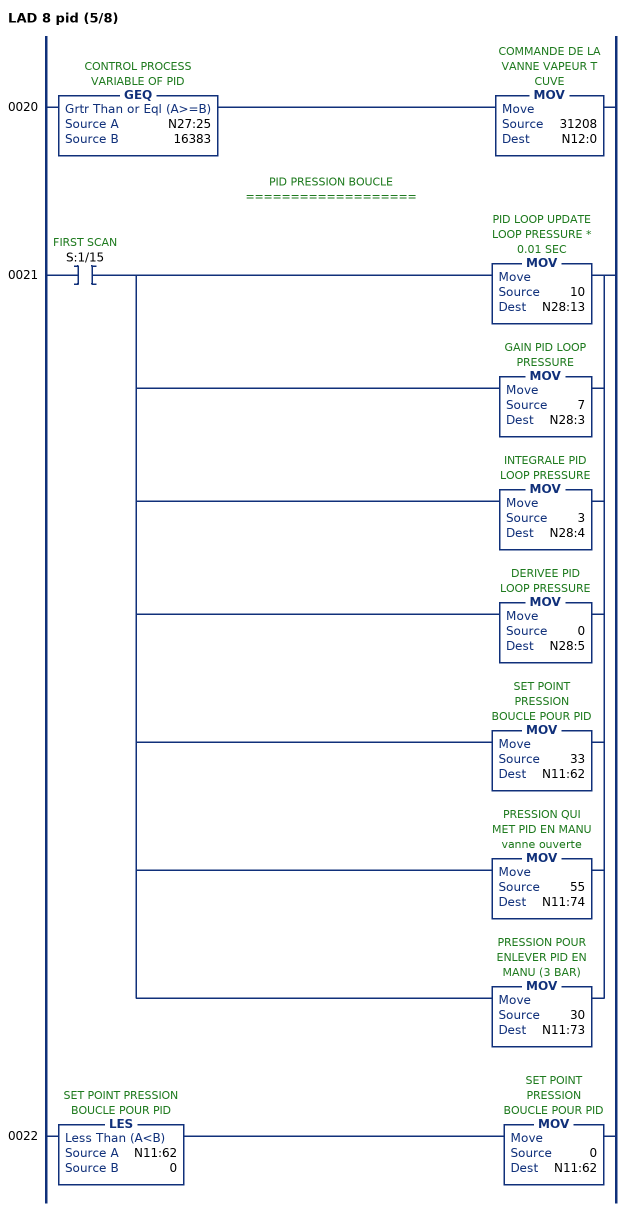
% Rung: 20 %
SOR GEQ N27:25 16383 MOV 31208 N12:0 EOR
%   N27:25  "CONTROL PROCESS VARIABLE OF PID" %
%   N12:0  "COMMANDE DE LA VANNE VAPEUR T CUVE" %
% Rung: 21 %
% PID PRESSION BOUCLE
% =================== %
SOR XIC S:1/15 BST MOV 10 N28:13 NXB MOV 7 N28:3 NXB MOV 3 N28:4 NXB MOV 0 N28:5 NXB MOV 33 N11:62 NXB MOV 55 N11:74 NXB MOV 30 N11:73 BND EOR
%   S:1/15  "FIRST SCAN" %
%   N28:13  "PID LOOP UPDATE LOOP PRESSURE * 0.01 SEC" %
%   N28:3  "GAIN PID LOOP PRESSURE" %
%   N28:4  "INTEGRALE PID LOOP PRESSURE" %
%   N28:5  "DERIVEE PID LOOP PRESSURE" %
%   N11:62  "SET POINT PRESSION BOUCLE POUR PID" %
%   N11:74  "PRESSION QUI MET PID EN MANU vanne ouverte" %
%   N11:73  "PRESSION POUR ENLEVER PID EN MANU (3 BAR)" %
% Rung: 22 %
SOR LES N11:62 0 MOV 0 N11:62 EOR
%   N11:62  "SET POINT PRESSION BOUCLE POUR PID" %

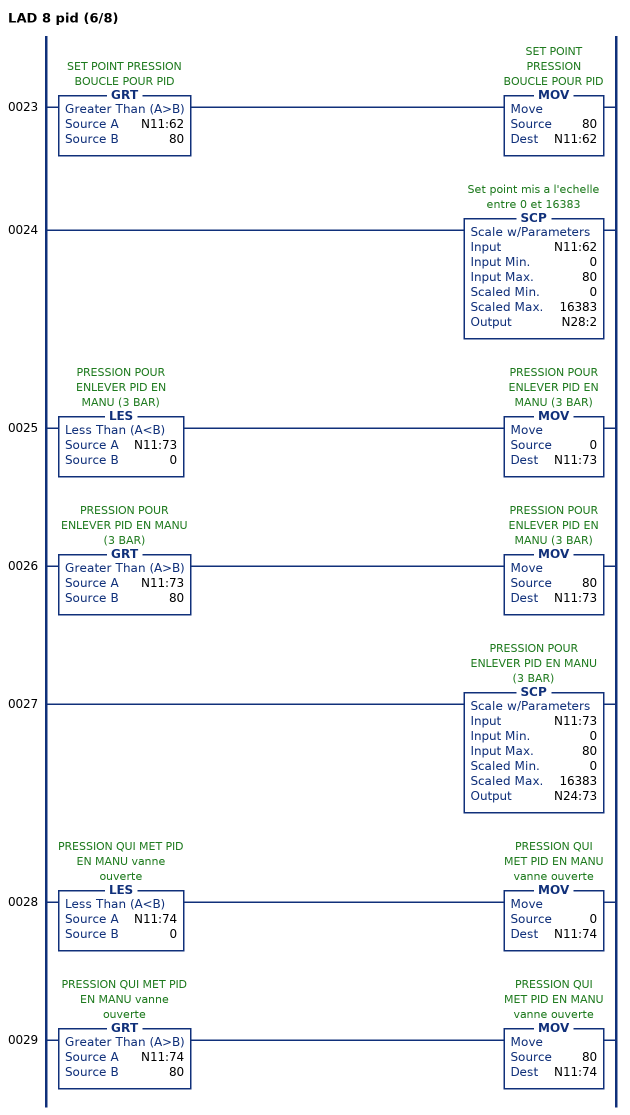
% Rung: 23 %
SOR GRT N11:62 80 MOV 80 N11:62 EOR
%   N11:62  "SET POINT PRESSION BOUCLE POUR PID" %
% Rung: 24 %
SOR SCP N11:62 0 80 0 16383 N28:2 EOR
%   N11:62  "SET POINT PRESSION BOUCLE POUR PID" %
%   N28:2  "Set point mis a l'echelle entre 0 et 16383" %
% Rung: 25 %
SOR LES N11:73 0 MOV 0 N11:73 EOR
%   N11:73  "PRESSION POUR ENLEVER PID EN MANU (3 BAR)" %
% Rung: 26 %
SOR GRT N11:73 80 MOV 80 N11:73 EOR
%   N11:73  "PRESSION POUR ENLEVER PID EN MANU (3 BAR)" %
% Rung: 27 %
SOR SCP N11:73 0 80 0 16383 N24:73 EOR
%   N11:73  "PRESSION POUR ENLEVER PID EN MANU (3 BAR)" %
%   N24:73  "PRESSION POUR ENLEVER PID EN MANU (3 BAR)" %
% Rung: 28 %
SOR LES N11:74 0 MOV 0 N11:74 EOR
%   N11:74  "PRESSION QUI MET PID EN MANU vanne ouverte" %
% Rung: 29 %
SOR GRT N11:74 80 MOV 80 N11:74 EOR
%   N11:74  "PRESSION QUI MET PID EN MANU vanne ouverte" %

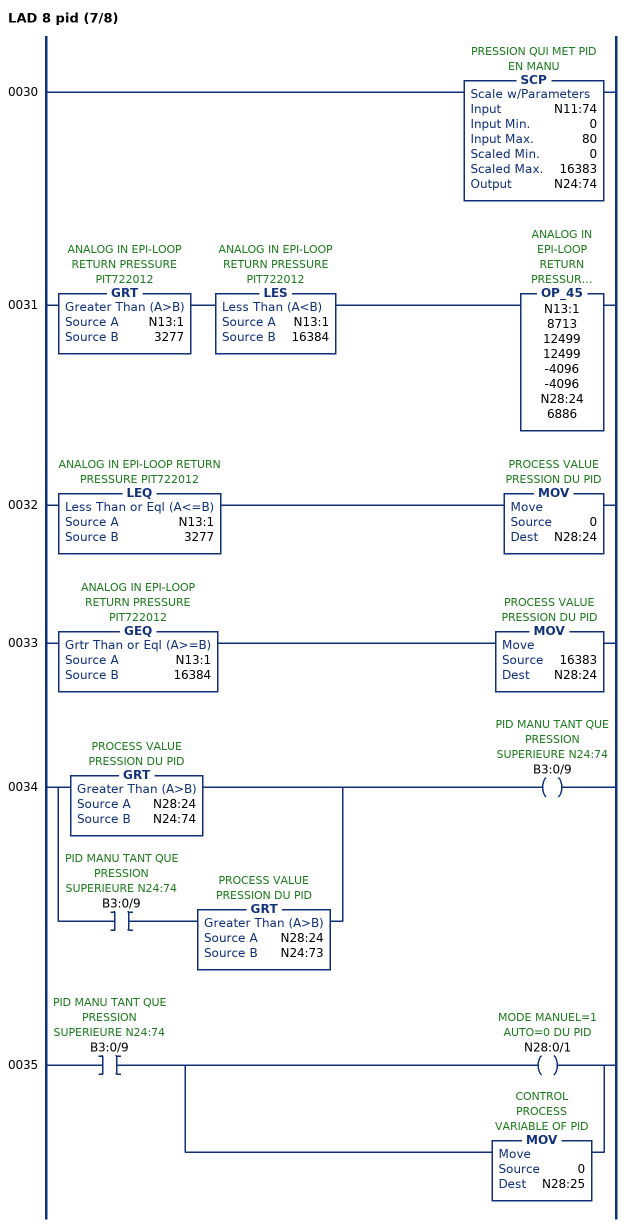
% Rung: 30 %
SOR SCP N11:74 0 80 0 16383 N24:74 EOR
%   N11:74  "PRESSION QUI MET PID EN MANU vanne ouverte" %
%   N24:74  "PRESSION QUI MET PID EN MANU" %
% Rung: 31 %
SOR GRT N13:1 3277 LES N13:1 16384 OP_45 N13:1 8713 12499 12499 -4096 -4096 N28:24 6886 EOR
%   N13:1  "ANALOG IN EPI-LOOP RETURN PRESSURE PIT722012" %
%   N28:24  "PROCESS VALUE PRESSION DU PID" %
% Rung: 32 %
SOR LEQ N13:1 3277 MOV 0 N28:24 EOR
%   N13:1  "ANALOG IN EPI-LOOP RETURN PRESSURE PIT722012" %
%   N28:24  "PROCESS VALUE PRESSION DU PID" %
% Rung: 33 %
SOR GEQ N13:1 16384 MOV 16383 N28:24 EOR
%   N13:1  "ANALOG IN EPI-LOOP RETURN PRESSURE PIT722012" %
%   N28:24  "PROCESS VALUE PRESSION DU PID" %
% Rung: 34 %
SOR BST GRT N28:24 N24:74 NXB XIC B3:0/9 GRT N28:24 N24:73 BND OTE B3:0/9 EOR
%   N28:24  "PROCESS VALUE PRESSION DU PID" %
%   N24:74  "PRESSION QUI MET PID EN MANU" %
%   B3:0/9  "PID MANU TANT QUE PRESSION SUPERIEURE N24:74" %
%   N24:73  "PRESSION POUR ENLEVER PID EN MANU (3 BAR)" %
% Rung: 35 %
SOR XIC B3:0/9 BST OTE N28:0/1 NXB MOV 0 N28:25 BND EOR
%   B3:0/9  "PID MANU TANT QUE PRESSION SUPERIEURE N24:74" %
%   N28:0/1  "MODE MANUEL=1 AUTO=0 DU PID" %
%   N28:25  "CONTROL PROCESS VARIABLE OF PID" %

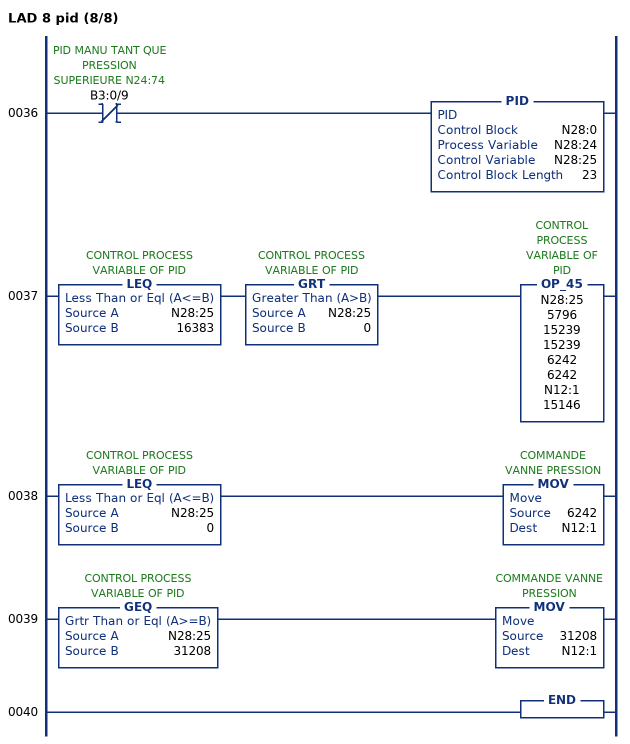
% Rung: 36 %
SOR XIO B3:0/9 PID N28:0 N28:24 N28:25 23 EOR
%   B3:0/9  "PID MANU TANT QUE PRESSION SUPERIEURE N24:74" %
%   N28:24  "PROCESS VALUE PRESSION DU PID" %
%   N28:25  "CONTROL PROCESS VARIABLE OF PID" %
% Rung: 37 %
SOR LEQ N28:25 16383 GRT N28:25 0 OP_45 N28:25 5796 15239 15239 6242 6242 N12:1 15146 EOR
%   N28:25  "CONTROL PROCESS VARIABLE OF PID" %
%   N12:1  "COMMANDE VANNE PRESSION" %
% Rung: 38 %
SOR LEQ N28:25 0 MOV 6242 N12:1 EOR
%   N28:25  "CONTROL PROCESS VARIABLE OF PID" %
%   N12:1  "COMMANDE VANNE PRESSION" %
% Rung: 39 %
SOR GEQ N28:25 31208 MOV 31208 N12:1 EOR
%   N28:25  "CONTROL PROCESS VARIABLE OF PID" %
%   N12:1  "COMMANDE VANNE PRESSION" %
% Rung: 40 %
SOR END EOR

LADDER 9 "affichage"
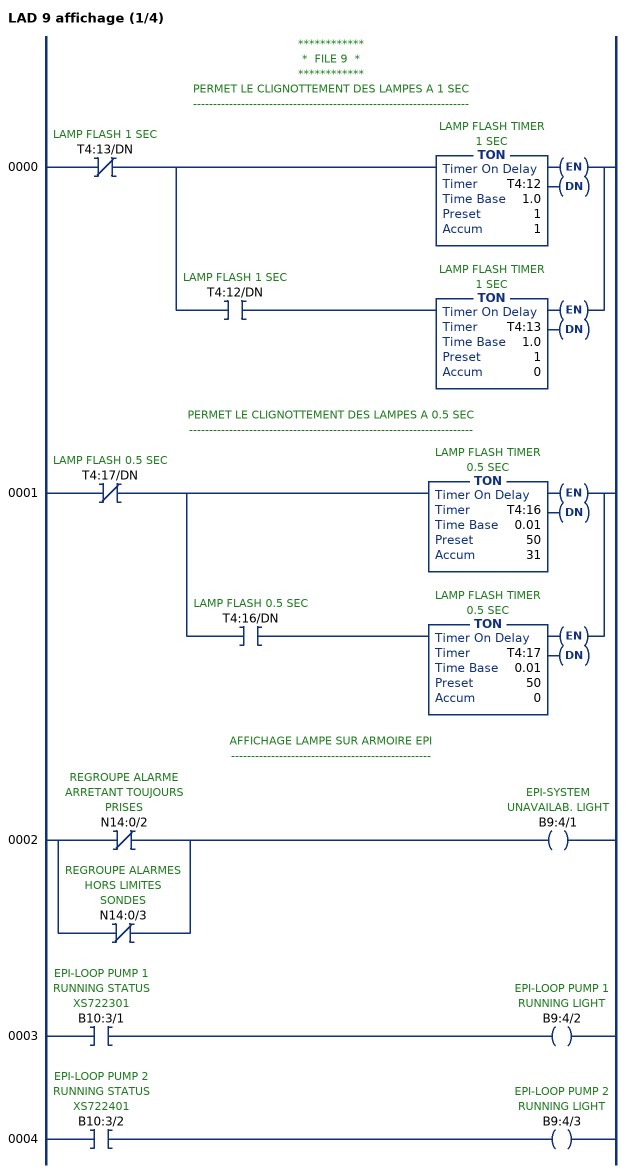
% Rung: 0 %
% ************
% *  FILE 9  *
% ************
% 
% PERMET LE CLIGNOTTEMENT DES LAMPES A 1 SEC
% --------------------------------------------------------------------- %
SOR XIO T4:13/DN BST TON T4:12 1.0 1 1 NXB XIC T4:12/DN TON T4:13 1.0 1 0 BND EOR
%   T4:13/DN  "LAMP FLASH 1 SEC" %
%   T4:12  "LAMP FLASH TIMER 1 SEC" %
%   T4:12/DN  "LAMP FLASH 1 SEC" %
%   T4:13  "LAMP FLASH TIMER 1 SEC" %
% Rung: 1 %
% PERMET LE CLIGNOTTEMENT DES LAMPES A 0.5 SEC
% ----------------------------------------------------------------------- %
SOR XIO T4:17/DN BST TON T4:16 0.01 50 31 NXB XIC T4:16/DN TON T4:17 0.01 50 0 BND EOR
%   T4:17/DN  "LAMP FLASH 0.5 SEC" %
%   T4:16  "LAMP FLASH TIMER 0.5 SEC" %
%   T4:16/DN  "LAMP FLASH 0.5 SEC" %
%   T4:17  "LAMP FLASH TIMER 0.5 SEC" %
% Rung: 2 %
% AFFICHAGE LAMPE SUR ARMOIRE EPI
% -------------------------------------------------- %
SOR BST XIO N14:0/2 NXB XIO N14:0/3 BND OTE B9:4/1 EOR
%   N14:0/2  "REGROUPE ALARME ARRETANT TOUJOURS PRISES" %
%   N14:0/3  "REGROUPE ALARMES HORS LIMITES SONDES" %
%   B9:4/1  "EPI-SYSTEM UNAVAILAB. LIGHT" %
% Rung: 3 %
SOR XIC B10:3/1 OTE B9:4/2 EOR
%   B10:3/1  "EPI-LOOP PUMP 1 RUNNING STATUS XS722301" %
%   B9:4/2  "EPI-LOOP PUMP 1 RUNNING LIGHT" %
% Rung: 4 %
SOR XIC B10:3/2 OTE B9:4/3 EOR
%   B10:3/2  "EPI-LOOP PUMP 2 RUNNING STATUS XS722401" %
%   B9:4/3  "EPI-LOOP PUMP 2 RUNNING LIGHT" %

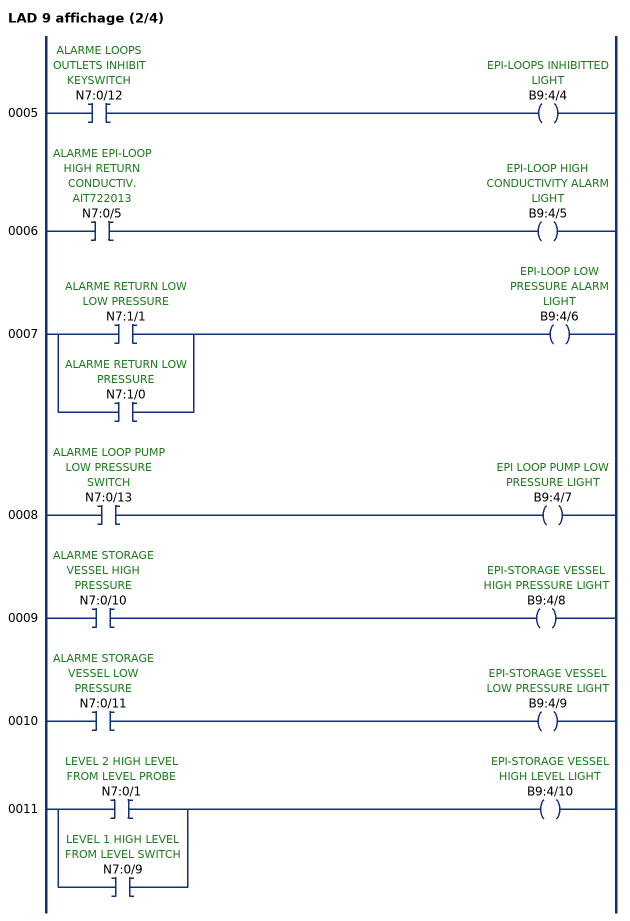
% Rung: 5 %
SOR XIC N7:0/12 OTE B9:4/4 EOR
%   N7:0/12  "ALARME LOOPS OUTLETS INHIBIT KEYSWITCH" %
%   B9:4/4  "EPI-LOOPS INHIBITTED LIGHT" %
% Rung: 6 %
SOR XIC N7:0/5 OTE B9:4/5 EOR
%   N7:0/5  "ALARME EPI-LOOP HIGH RETURN CONDUCTIV. AIT722013" %
%   B9:4/5  "EPI-LOOP HIGH CONDUCTIVITY ALARM LIGHT" %
% Rung: 7 %
SOR BST XIC N7:1/1 NXB XIC N7:1/0 BND OTE B9:4/6 EOR
%   N7:1/1  "ALARME RETURN LOW LOW PRESSURE" %
%   N7:1/0  "ALARME RETURN LOW PRESSURE" %
%   B9:4/6  "EPI-LOOP LOW PRESSURE ALARM LIGHT" %
% Rung: 8 %
SOR XIC N7:0/13 OTE B9:4/7 EOR
%   N7:0/13  "ALARME LOOP PUMP LOW PRESSURE SWITCH" %
%   B9:4/7  "EPI LOOP PUMP LOW PRESSURE LIGHT" %
% Rung: 9 %
SOR XIC N7:0/10 OTE B9:4/8 EOR
%   N7:0/10  "ALARME STORAGE VESSEL HIGH PRESSURE" %
%   B9:4/8  "EPI-STORAGE VESSEL HIGH PRESSURE LIGHT" %
% Rung: 10 %
SOR XIC N7:0/11 OTE B9:4/9 EOR
%   N7:0/11  "ALARME STORAGE VESSEL LOW PRESSURE" %
%   B9:4/9  "EPI-STORAGE VESSEL LOW PRESSURE LIGHT" %
% Rung: 11 %
SOR BST XIC N7:0/1 NXB XIC N7:0/9 BND OTE B9:4/10 EOR
%   N7:0/1  "LEVEL 2 HIGH LEVEL FROM LEVEL PROBE" %
%   N7:0/9  "LEVEL 1 HIGH LEVEL FROM LEVEL SWITCH" %
%   B9:4/10  "EPI-STORAGE VESSEL HIGH LEVEL LIGHT" %

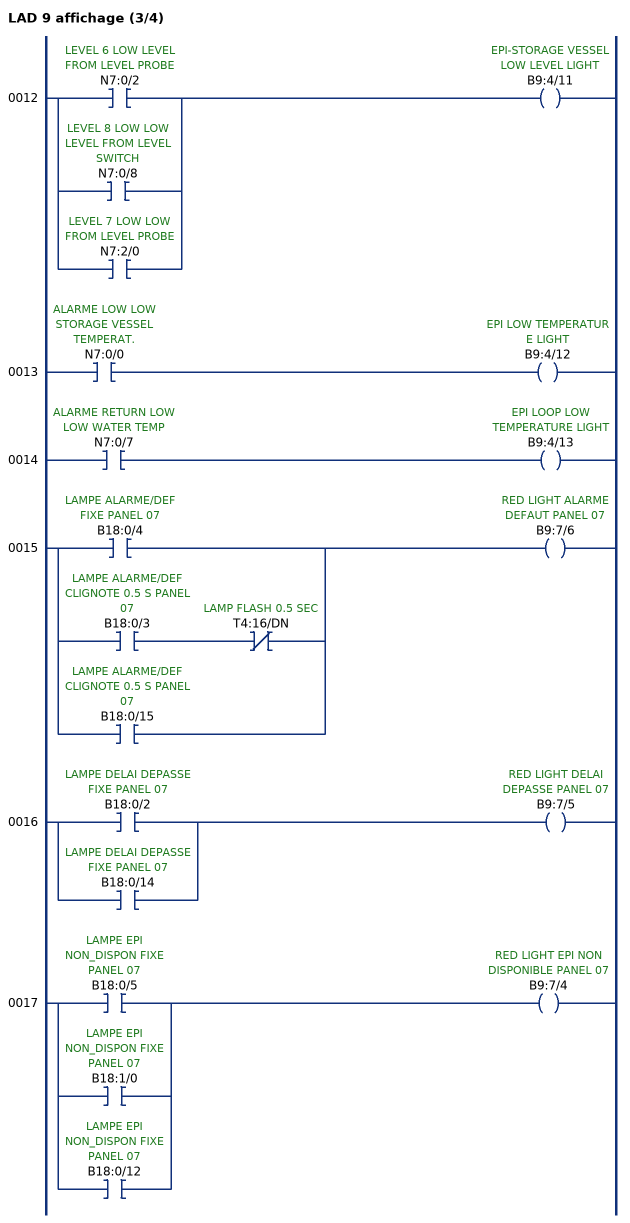
% Rung: 12 %
SOR BST XIC N7:0/2 NXB XIC N7:0/8 NXB XIC N7:2/0 BND OTE B9:4/11 EOR
%   N7:0/2  "LEVEL 6 LOW LEVEL FROM LEVEL PROBE" %
%   N7:0/8  "LEVEL 8 LOW LOW LEVEL FROM LEVEL SWITCH" %
%   N7:2/0  "LEVEL 7 LOW LOW FROM LEVEL PROBE" %
%   B9:4/11  "EPI-STORAGE VESSEL LOW LEVEL LIGHT" %
% Rung: 13 %
SOR XIC N7:0/0 OTE B9:4/12 EOR
%   N7:0/0  "ALARME LOW LOW STORAGE VESSEL TEMPERAT." %
%   B9:4/12  "EPI LOW TEMPERATURE LIGHT" %
% Rung: 14 %
SOR XIC N7:0/7 OTE B9:4/13 EOR
%   N7:0/7  "ALARME RETURN LOW LOW WATER TEMP" %
%   B9:4/13  "EPI LOOP LOW TEMPERATURE LIGHT" %
% Rung: 15 %
SOR BST XIC B18:0/4 NXB XIC B18:0/3 XIO T4:16/DN NXB XIC B18:0/15 BND OTE B9:7/6 EOR
%   B18:0/4  "LAMPE ALARME/DEF FIXE PANEL 07" %
%   B18:0/3  "LAMPE ALARME/DEF CLIGNOTE 0.5 S PANEL 07" %
%   T4:16/DN  "LAMP FLASH 0.5 SEC" %
%   B18:0/15  "LAMPE ALARME/DEF CLIGNOTE 0.5 S PANEL 07" %
%   B9:7/6  "RED LIGHT ALARME DEFAUT PANEL 07" %
% Rung: 16 %
SOR BST XIC B18:0/2 NXB XIC B18:0/14 BND OTE B9:7/5 EOR
%   B18:0/2  "LAMPE DELAI DEPASSE FIXE PANEL 07" %
%   B18:0/14  "LAMPE DELAI DEPASSE FIXE PANEL 07" %
%   B9:7/5  "RED LIGHT DELAI DEPASSE PANEL 07" %
% Rung: 17 %
SOR BST XIC B18:0/5 NXB XIC B18:1/0 NXB XIC B18:0/12 BND OTE B9:7/4 EOR
%   B18:0/5  "LAMPE EPI NON_DISPON FIXE PANEL 07" %
%   B18:1/0  "LAMPE EPI NON_DISPON FIXE PANEL 07" %
%   B18:0/12  "LAMPE EPI NON_DISPON FIXE PANEL 07" %
%   B9:7/4  "RED LIGHT EPI NON DISPONIBLE PANEL 07" %

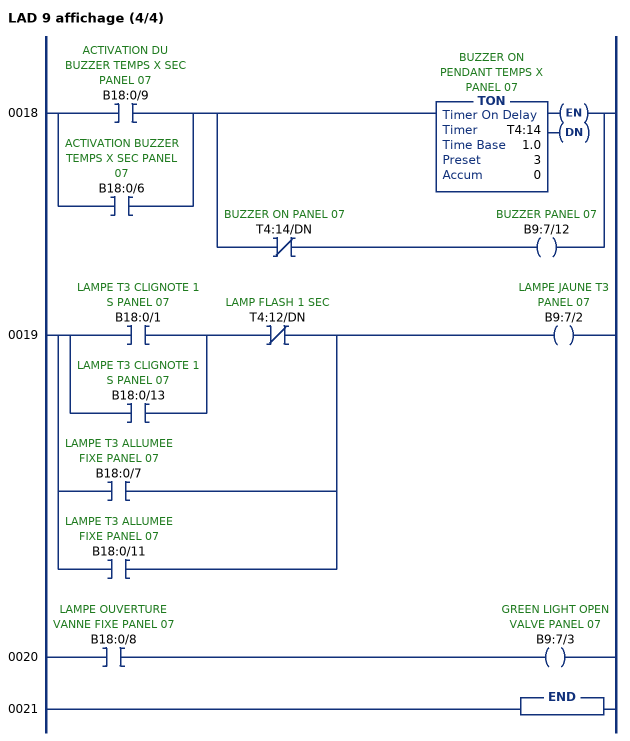
% Rung: 18 %
SOR BST XIC B18:0/9 NXB XIC B18:0/6 BND BST TON T4:14 1.0 3 0 NXB XIO T4:14/DN OTE B9:7/12 BND EOR
%   B18:0/9  "ACTIVATION DU BUZZER TEMPS X SEC PANEL 07" %
%   B18:0/6  "ACTIVATION BUZZER TEMPS X SEC PANEL 07" %
%   T4:14  "BUZZER ON PENDANT TEMPS X PANEL 07" %
%   T4:14/DN  "BUZZER ON PANEL 07" %
%   B9:7/12  "BUZZER PANEL 07" %
% Rung: 19 %
SOR BST BST XIC B18:0/1 NXB XIC B18:0/13 BND XIO T4:12/DN NXB XIC B18:0/7 NXB XIC B18:0/11 BND OTE B9:7/2 EOR
%   B18:0/1  "LAMPE T3 CLIGNOTE 1 S PANEL 07" %
%   B18:0/13  "LAMPE T3 CLIGNOTE 1 S PANEL 07" %
%   T4:12/DN  "LAMP FLASH 1 SEC" %
%   B18:0/7  "LAMPE T3 ALLUMEE FIXE PANEL 07" %
%   B18:0/11  "LAMPE T3 ALLUMEE FIXE PANEL 07" %
%   B9:7/2  "LAMPE JAUNE T3 PANEL 07" %
% Rung: 20 %
SOR XIC B18:0/8 OTE B9:7/3 EOR
%   B18:0/8  "LAMPE OUVERTURE VANNE FIXE PANEL 07" %
%   B9:7/3  "GREEN LIGHT OPEN VALVE PANEL 07" %
% Rung: 21 %
SOR END EOR

LADDER 10 "table_sort"
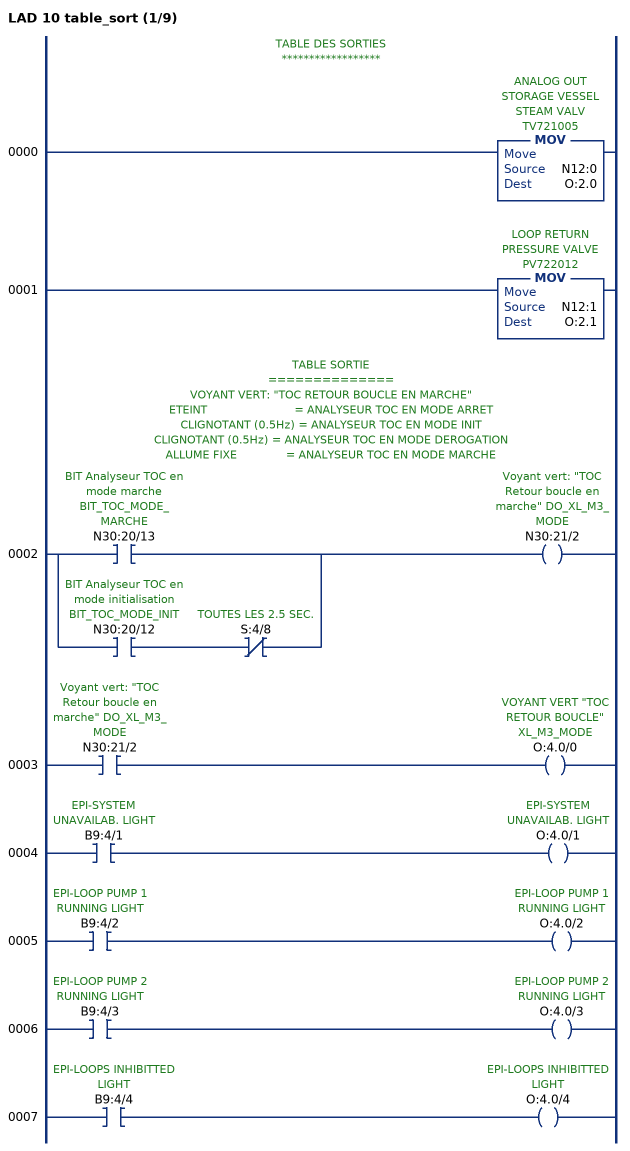
% Rung: 0 %
% TABLE DES SORTIES
% ****************** %
SOR MOV N12:0 O:2.0 EOR
%   N12:0  "COMMANDE DE LA VANNE VAPEUR T CUVE" %
%   O:2.0  "ANALOG OUT STORAGE VESSEL STEAM VALV TV721005" %
% Rung: 1 %
SOR MOV N12:1 O:2.1 EOR
%   N12:1  "COMMANDE VANNE PRESSION" %
%   O:2.1  "LOOP RETURN PRESSURE VALVE PV722012" %
% Rung: 2 %
% TABLE SORTIE
% ==============
% VOYANT VERT: "TOC RETOUR BOUCLE EN MARCHE"
% 
% ETEINT                         = ANALYSEUR TOC EN MODE ARRET
% CLIGNOTANT (0.5Hz) = ANALYSEUR TOC EN MODE INIT
% CLIGNOTANT (0.5Hz) = ANALYSEUR TOC EN MODE DEROGATION
% ALLUME FIXE              = ANALYSEUR TOC EN MODE MARCHE %
SOR BST XIC N30:20/13 NXB XIC N30:20/12 XIO S:4/8 BND OTE N30:21/2 EOR
%   N30:20/13  BIT_TOC_MODE_MARCHE  "BIT Analyseur TOC en mode marche" %
%   N30:20/12  BIT_TOC_MODE_INIT  "BIT Analyseur TOC en mode initialisation" %
%   S:4/8  "TOUTES LES 2.5 SEC." %
%   N30:21/2  DO_XL_M3_MODE  "Voyant vert: "TOC Retour boucle en marche"" %
% Rung: 3 %
SOR XIC N30:21/2 OTE O:4.0/0 EOR
%   N30:21/2  DO_XL_M3_MODE  "Voyant vert: "TOC Retour boucle en marche"" %
%   O:4.0/0  XL_M3_MODE  "VOYANT VERT "TOC RETOUR BOUCLE"" %
% Rung: 4 %
SOR XIC B9:4/1 OTE O:4.0/1 EOR
%   B9:4/1  "EPI-SYSTEM UNAVAILAB. LIGHT" %
%   O:4.0/1  "EPI-SYSTEM UNAVAILAB. LIGHT" %
% Rung: 5 %
SOR XIC B9:4/2 OTE O:4.0/2 EOR
%   B9:4/2  "EPI-LOOP PUMP 1 RUNNING LIGHT" %
%   O:4.0/2  "EPI-LOOP PUMP 1 RUNNING LIGHT" %
% Rung: 6 %
SOR XIC B9:4/3 OTE O:4.0/3 EOR
%   B9:4/3  "EPI-LOOP PUMP 2 RUNNING LIGHT" %
%   O:4.0/3  "EPI-LOOP PUMP 2 RUNNING LIGHT" %
% Rung: 7 %
SOR XIC B9:4/4 OTE O:4.0/4 EOR
%   B9:4/4  "EPI-LOOPS INHIBITTED LIGHT" %
%   O:4.0/4  "EPI-LOOPS INHIBITTED LIGHT" %

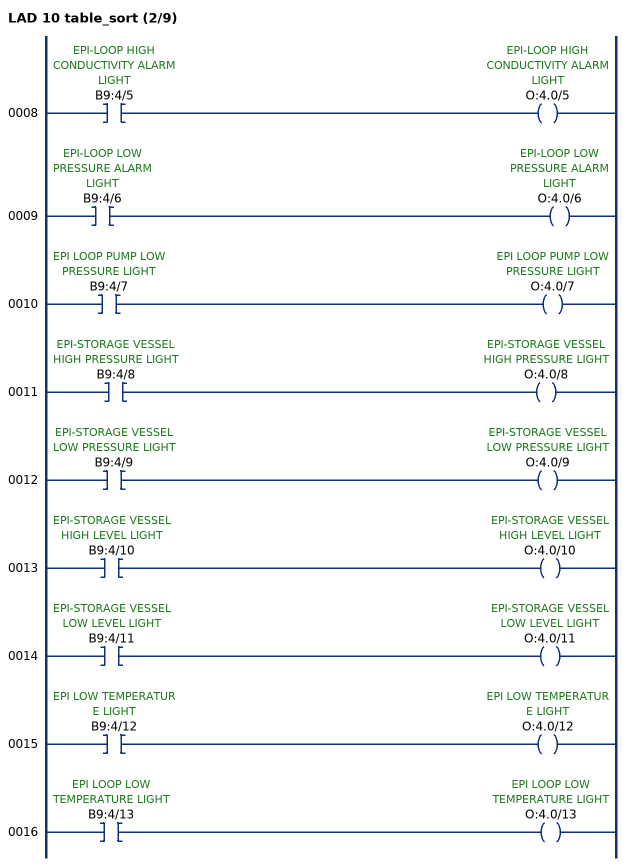
% Rung: 8 %
SOR XIC B9:4/5 OTE O:4.0/5 EOR
%   B9:4/5  "EPI-LOOP HIGH CONDUCTIVITY ALARM LIGHT" %
%   O:4.0/5  "EPI-LOOP HIGH CONDUCTIVITY ALARM LIGHT" %
% Rung: 9 %
SOR XIC B9:4/6 OTE O:4.0/6 EOR
%   B9:4/6  "EPI-LOOP LOW PRESSURE ALARM LIGHT" %
%   O:4.0/6  "EPI-LOOP LOW PRESSURE ALARM LIGHT" %
% Rung: 10 %
SOR XIC B9:4/7 OTE O:4.0/7 EOR
%   B9:4/7  "EPI LOOP PUMP LOW PRESSURE LIGHT" %
%   O:4.0/7  "EPI LOOP PUMP LOW PRESSURE LIGHT" %
% Rung: 11 %
SOR XIC B9:4/8 OTE O:4.0/8 EOR
%   B9:4/8  "EPI-STORAGE VESSEL HIGH PRESSURE LIGHT" %
%   O:4.0/8  "EPI-STORAGE VESSEL HIGH PRESSURE LIGHT" %
% Rung: 12 %
SOR XIC B9:4/9 OTE O:4.0/9 EOR
%   B9:4/9  "EPI-STORAGE VESSEL LOW PRESSURE LIGHT" %
%   O:4.0/9  "EPI-STORAGE VESSEL LOW PRESSURE LIGHT" %
% Rung: 13 %
SOR XIC B9:4/10 OTE O:4.0/10 EOR
%   B9:4/10  "EPI-STORAGE VESSEL HIGH LEVEL LIGHT" %
%   O:4.0/10  "EPI-STORAGE VESSEL HIGH LEVEL LIGHT" %
% Rung: 14 %
SOR XIC B9:4/11 OTE O:4.0/11 EOR
%   B9:4/11  "EPI-STORAGE VESSEL LOW LEVEL LIGHT" %
%   O:4.0/11  "EPI-STORAGE VESSEL LOW LEVEL LIGHT" %
% Rung: 15 %
SOR XIC B9:4/12 OTE O:4.0/12 EOR
%   B9:4/12  "EPI LOW TEMPERATURE LIGHT" %
%   O:4.0/12  "EPI LOW TEMPERATURE LIGHT" %
% Rung: 16 %
SOR XIC B9:4/13 OTE O:4.0/13 EOR
%   B9:4/13  "EPI LOOP LOW TEMPERATURE LIGHT" %
%   O:4.0/13  "EPI LOOP LOW TEMPERATURE LIGHT" %

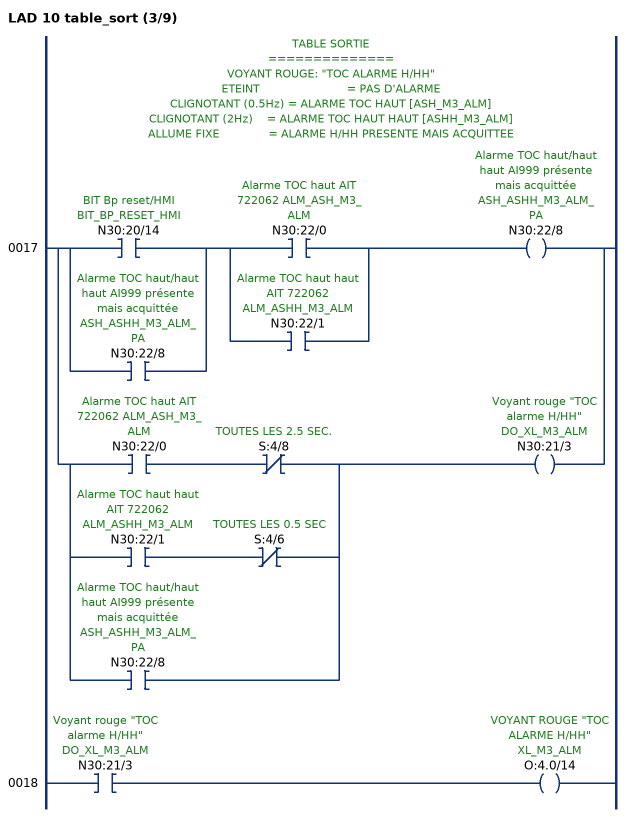
% Rung: 17 %
% TABLE SORTIE
% ==============
% VOYANT ROUGE: "TOC ALARME H/HH"
% 
% ETEINT                         = PAS D'ALARME
% CLIGNOTANT (0.5Hz) = ALARME TOC HAUT [ASH_M3_ALM]
% CLIGNOTANT (2Hz)    = ALARME TOC HAUT HAUT [ASHH_M3_ALM]
% ALLUME FIXE              = ALARME H/HH PRESENTE MAIS ACQUITTEE %
SOR BST BST XIC N30:20/14 NXB XIC N30:22/8 BND BST XIC N30:22/0 NXB XIC N30:22/1 BND OTE N30:22/8 NXB BST XIC N30:22/0 XIO S:4/8 NXB XIC N30:22/1 XIO S:4/6 NXB XIC N30:22/8 BND OTE N30:21/3 BND EOR
%   N30:20/14  BIT_BP_RESET_HMI  "BIT Bp reset/HMI" %
%   N30:22/8  ASH_ASHH_M3_ALM_PA  "Alarme TOC haut/haut haut AI999 présente mais acquittée" %
%   N30:22/0  ALM_ASH_M3_ALM  "Alarme TOC haut AIT 722062" %
%   N30:22/1  ALM_ASHH_M3_ALM  "Alarme TOC haut haut AIT 722062" %
%   S:4/8  "TOUTES LES 2.5 SEC." %
%   S:4/6  "TOUTES LES 0.5 SEC" %
%   N30:21/3  DO_XL_M3_ALM  "Voyant rouge "TOC alarme H/HH"" %
% Rung: 18 %
SOR XIC N30:21/3 OTE O:4.0/14 EOR
%   N30:21/3  DO_XL_M3_ALM  "Voyant rouge "TOC alarme H/HH"" %
%   O:4.0/14  XL_M3_ALM  "VOYANT ROUGE "TOC ALARME H/HH"" %

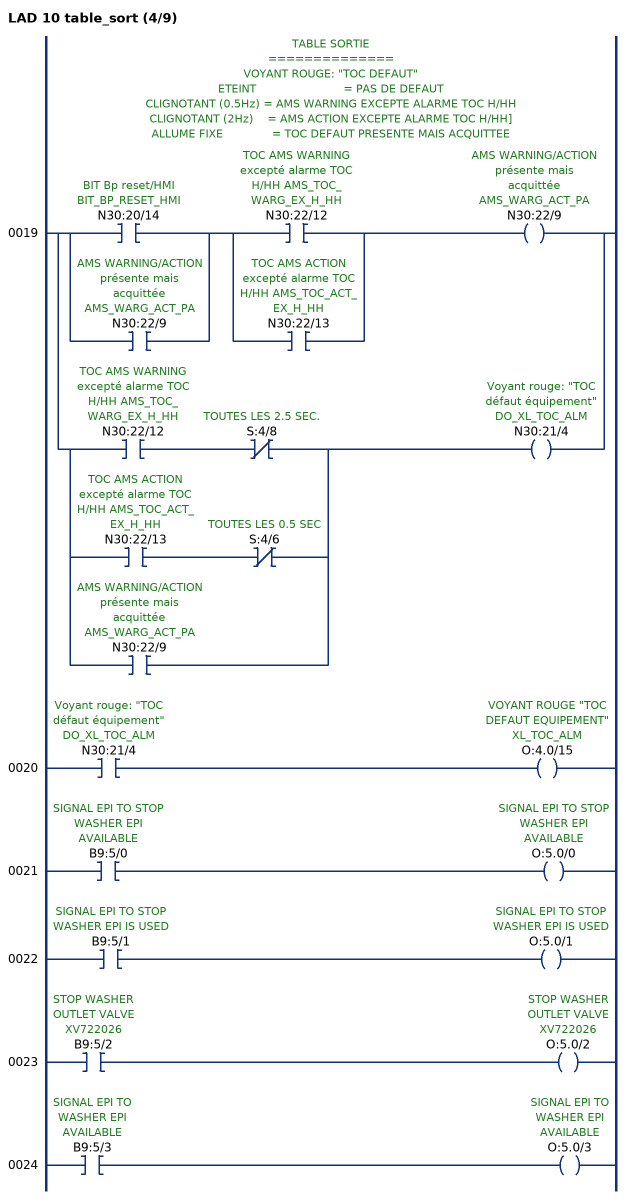
% Rung: 19 %
% TABLE SORTIE
% ==============
% VOYANT ROUGE: "TOC DEFAUT"
% 
% ETEINT                         = PAS DE DEFAUT
% CLIGNOTANT (0.5Hz) = AMS WARNING EXCEPTE ALARME TOC H/HH
% CLIGNOTANT (2Hz)    = AMS ACTION EXCEPTE ALARME TOC H/HH]
% ALLUME FIXE              = TOC DEFAUT PRESENTE MAIS ACQUITTEE %
SOR BST BST XIC N30:20/14 NXB XIC N30:22/9 BND BST XIC N30:22/12 NXB XIC N30:22/13 BND OTE N30:22/9 NXB BST XIC N30:22/12 XIO S:4/8 NXB XIC N30:22/13 XIO S:4/6 NXB XIC N30:22/9 BND OTE N30:21/4 BND EOR
%   N30:20/14  BIT_BP_RESET_HMI  "BIT Bp reset/HMI" %
%   N30:22/9  AMS_WARG_ACT_PA  "AMS WARNING/ACTION présente mais acquittée" %
%   N30:22/12  AMS_TOC_WARG_EX_H_HH  "TOC AMS WARNING excepté alarme TOC H/HH" %
%   N30:22/13  AMS_TOC_ACT_EX_H_HH  "TOC AMS ACTION excepté alarme TOC H/HH" %
%   S:4/8  "TOUTES LES 2.5 SEC." %
%   S:4/6  "TOUTES LES 0.5 SEC" %
%   N30:21/4  DO_XL_TOC_ALM  "Voyant rouge: "TOC défaut équipement"" %
% Rung: 20 %
SOR XIC N30:21/4 OTE O:4.0/15 EOR
%   N30:21/4  DO_XL_TOC_ALM  "Voyant rouge: "TOC défaut équipement"" %
%   O:4.0/15  XL_TOC_ALM  "VOYANT ROUGE "TOC DEFAUT EQUIPEMENT"" %
% Rung: 21 %
SOR XIC B9:5/0 OTE O:5.0/0 EOR
%   B9:5/0  "SIGNAL EPI TO STOP WASHER EPI AVAILABLE" %
%   O:5.0/0  "SIGNAL EPI TO STOP WASHER EPI AVAILABLE" %
% Rung: 22 %
SOR XIC B9:5/1 OTE O:5.0/1 EOR
%   B9:5/1  "SIGNAL EPI TO STOP WASHER EPI IS USED" %
%   O:5.0/1  "SIGNAL EPI TO STOP WASHER EPI IS USED" %
% Rung: 23 %
SOR XIC B9:5/2 OTE O:5.0/2 EOR
%   B9:5/2  "STOP WASHER OUTLET VALVE XV722026" %
%   O:5.0/2  "STOP WASHER OUTLET VALVE XV722026" %
% Rung: 24 %
SOR XIC B9:5/3 OTE O:5.0/3 EOR
%   B9:5/3  "SIGNAL EPI TO WASHER EPI AVAILABLE" %
%   O:5.0/3  "SIGNAL EPI TO WASHER EPI AVAILABLE" %

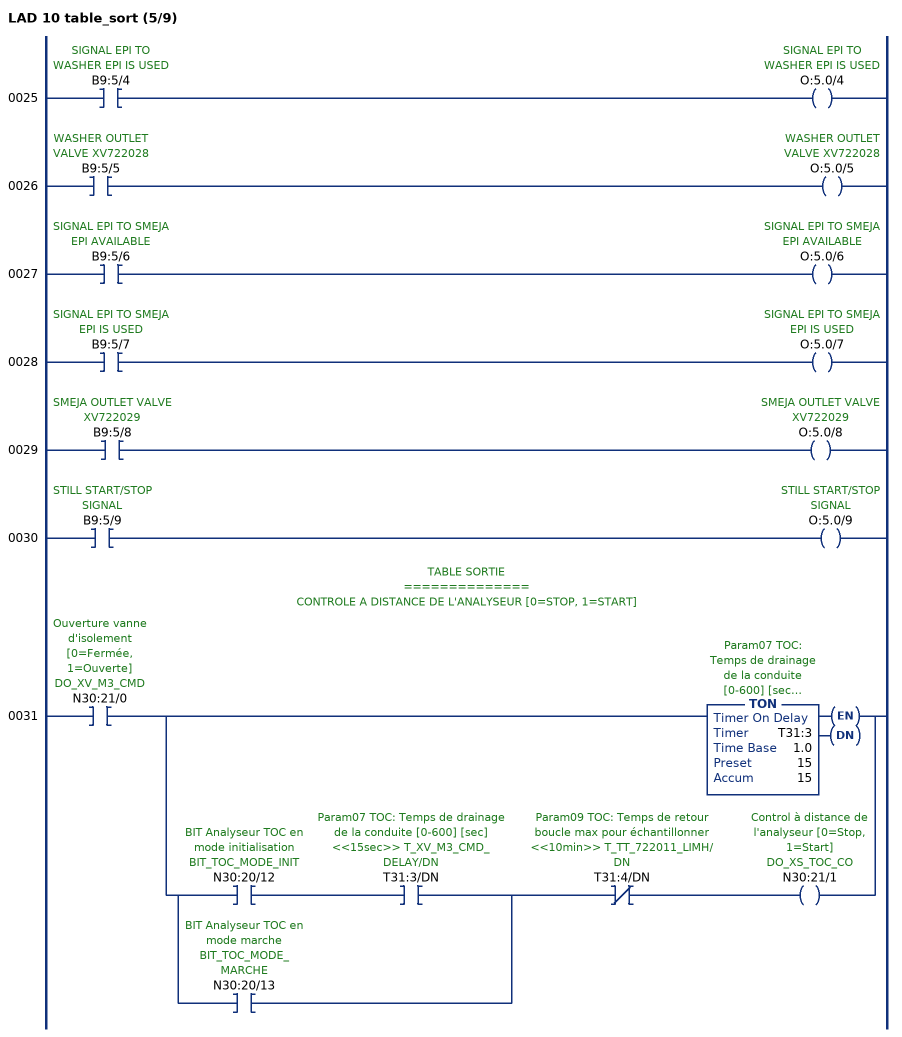
% Rung: 25 %
SOR XIC B9:5/4 OTE O:5.0/4 EOR
%   B9:5/4  "SIGNAL EPI TO WASHER EPI IS USED" %
%   O:5.0/4  "SIGNAL EPI TO WASHER EPI IS USED" %
% Rung: 26 %
SOR XIC B9:5/5 OTE O:5.0/5 EOR
%   B9:5/5  "WASHER OUTLET VALVE XV722028" %
%   O:5.0/5  "WASHER OUTLET VALVE XV722028" %
% Rung: 27 %
SOR XIC B9:5/6 OTE O:5.0/6 EOR
%   B9:5/6  "SIGNAL EPI TO SMEJA EPI AVAILABLE" %
%   O:5.0/6  "SIGNAL EPI TO SMEJA EPI AVAILABLE" %
% Rung: 28 %
SOR XIC B9:5/7 OTE O:5.0/7 EOR
%   B9:5/7  "SIGNAL EPI TO SMEJA EPI IS USED" %
%   O:5.0/7  "SIGNAL EPI TO SMEJA EPI IS USED" %
% Rung: 29 %
SOR XIC B9:5/8 OTE O:5.0/8 EOR
%   B9:5/8  "SMEJA OUTLET VALVE XV722029" %
%   O:5.0/8  "SMEJA OUTLET VALVE XV722029" %
% Rung: 30 %
SOR XIC B9:5/9 OTE O:5.0/9 EOR
%   B9:5/9  "STILL START/STOP SIGNAL" %
%   O:5.0/9  "STILL START/STOP SIGNAL" %
% Rung: 31 %
% TABLE SORTIE
% ==============
% CONTROLE A DISTANCE DE L'ANALYSEUR [0=STOP, 1=START] %
SOR XIC N30:21/0 BST TON T31:3 1.0 15 15 NXB BST XIC N30:20/12 XIC T31:3/DN NXB XIC N30:20/13 BND XIO T31:4/DN OTE N30:21/1 BND EOR
%   N30:21/0  DO_XV_M3_CMD  "Ouverture vanne d'isolement [0=Fermée, 1=Ouverte]" %
%   T31:3  T_XV_M3_CMD_DELAY  "Param07 TOC: Temps de drainage de la conduite [0-600] [sec] <<15sec>>" %
%   N30:20/12  BIT_TOC_MODE_INIT  "BIT Analyseur TOC en mode initialisation" %
%   N30:20/13  BIT_TOC_MODE_MARCHE  "BIT Analyseur TOC en mode marche" %
%   T31:4  T_TT_722011_LIMH  "Param09 TOC: Temps de retour boucle max pour échantillonner <<10min>>" %
%   N30:21/1  DO_XS_TOC_CO  "Control à distance de l'analyseur [0=Stop, 1=Start]" %

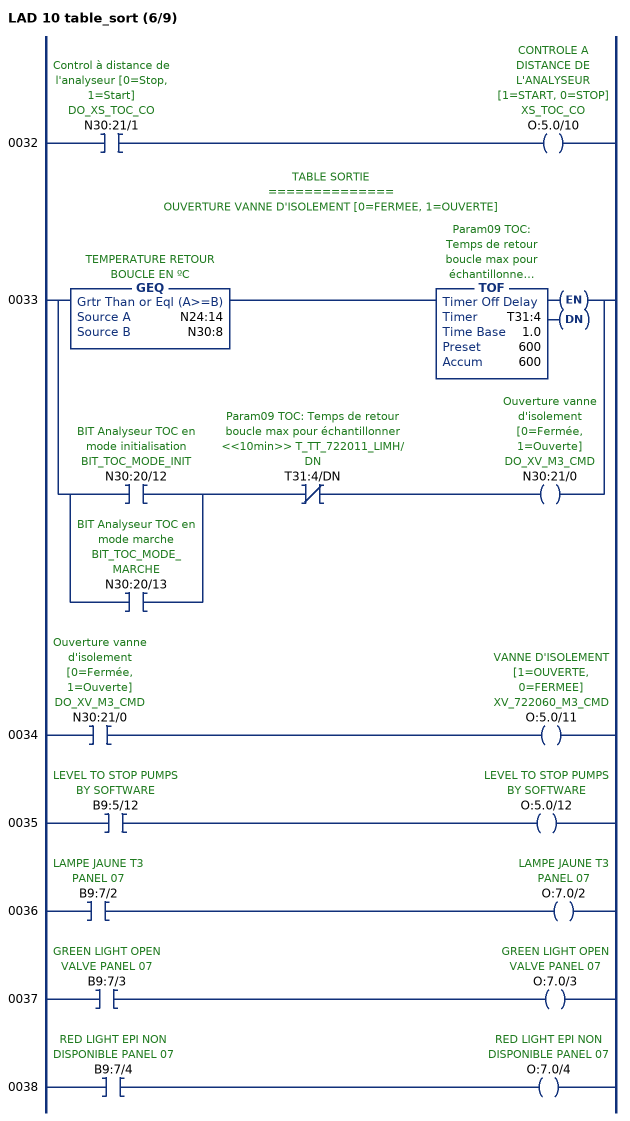
% Rung: 32 %
SOR XIC N30:21/1 OTE O:5.0/10 EOR
%   N30:21/1  DO_XS_TOC_CO  "Control à distance de l'analyseur [0=Stop, 1=Start]" %
%   O:5.0/10  XS_TOC_CO  "CONTROLE A DISTANCE DE L'ANALYSEUR [1=START, 0=STOP]" %
% Rung: 33 %
% TABLE SORTIE
% ==============
% OUVERTURE VANNE D'ISOLEMENT [0=FERMEE, 1=OUVERTE] %
SOR BST GEQ N24:14 N30:8 TOF T31:4 1.0 600 600 NXB BST XIC N30:20/12 NXB XIC N30:20/13 BND XIO T31:4/DN OTE N30:21/0 BND EOR
%   N24:14  "TEMPERATURE RETOUR BOUCLE EN ºC" %
%   N30:8  AI_TT_722011_LIMH  "Param08 TOC: Temp.de retour boucle max pour échantillonner [0-100] [°C] <<98°C>>" %
%   T31:4  T_TT_722011_LIMH  "Param09 TOC: Temps de retour boucle max pour échantillonner <<10min>>" %
%   N30:20/12  BIT_TOC_MODE_INIT  "BIT Analyseur TOC en mode initialisation" %
%   N30:20/13  BIT_TOC_MODE_MARCHE  "BIT Analyseur TOC en mode marche" %
%   N30:21/0  DO_XV_M3_CMD  "Ouverture vanne d'isolement [0=Fermée, 1=Ouverte]" %
% Rung: 34 %
SOR XIC N30:21/0 OTE O:5.0/11 EOR
%   N30:21/0  DO_XV_M3_CMD  "Ouverture vanne d'isolement [0=Fermée, 1=Ouverte]" %
%   O:5.0/11  XV_722060_M3_CMD  "VANNE D'ISOLEMENT [1=OUVERTE, 0=FERMEE]" %
% Rung: 35 %
SOR XIC B9:5/12 OTE O:5.0/12 EOR
%   B9:5/12  "LEVEL TO STOP PUMPS BY SOFTWARE" %
%   O:5.0/12  "LEVEL TO STOP PUMPS BY SOFTWARE" %
% Rung: 36 %
SOR XIC B9:7/2 OTE O:7.0/2 EOR
%   B9:7/2  "LAMPE JAUNE T3 PANEL 07" %
%   O:7.0/2  "LAMPE JAUNE T3 PANEL 07" %
% Rung: 37 %
SOR XIC B9:7/3 OTE O:7.0/3 EOR
%   B9:7/3  "GREEN LIGHT OPEN VALVE PANEL 07" %
%   O:7.0/3  "GREEN LIGHT OPEN VALVE PANEL 07" %
% Rung: 38 %
SOR XIC B9:7/4 OTE O:7.0/4 EOR
%   B9:7/4  "RED LIGHT EPI NON DISPONIBLE PANEL 07" %
%   O:7.0/4  "RED LIGHT EPI NON DISPONIBLE PANEL 07" %

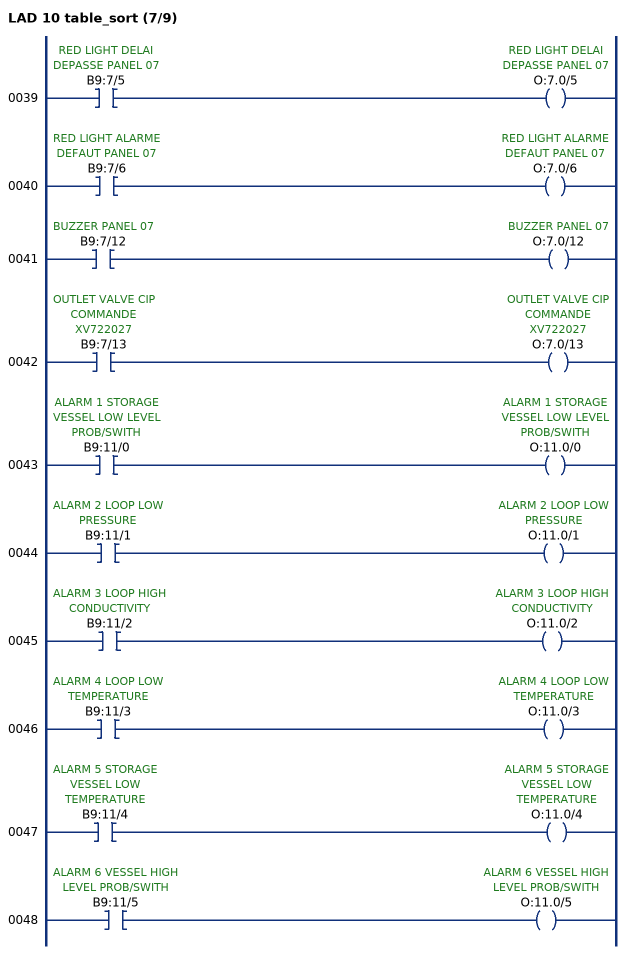
% Rung: 39 %
SOR XIC B9:7/5 OTE O:7.0/5 EOR
%   B9:7/5  "RED LIGHT DELAI DEPASSE PANEL 07" %
%   O:7.0/5  "RED LIGHT DELAI DEPASSE PANEL 07" %
% Rung: 40 %
SOR XIC B9:7/6 OTE O:7.0/6 EOR
%   B9:7/6  "RED LIGHT ALARME DEFAUT PANEL 07" %
%   O:7.0/6  "RED LIGHT ALARME DEFAUT PANEL 07" %
% Rung: 41 %
SOR XIC B9:7/12 OTE O:7.0/12 EOR
%   B9:7/12  "BUZZER PANEL 07" %
%   O:7.0/12  "BUZZER PANEL 07" %
% Rung: 42 %
SOR XIC B9:7/13 OTE O:7.0/13 EOR
%   B9:7/13  "OUTLET VALVE CIP COMMANDE XV722027" %
%   O:7.0/13  "OUTLET VALVE CIP COMMANDE XV722027" %
% Rung: 43 %
SOR XIC B9:11/0 OTE O:11.0/0 EOR
%   B9:11/0  "ALARM 1 STORAGE VESSEL LOW LEVEL PROB/SWITH" %
%   O:11.0/0  "ALARM 1 STORAGE VESSEL LOW LEVEL PROB/SWITH" %
% Rung: 44 %
SOR XIC B9:11/1 OTE O:11.0/1 EOR
%   B9:11/1  "ALARM 2 LOOP LOW PRESSURE" %
%   O:11.0/1  "ALARM 2 LOOP LOW PRESSURE" %
% Rung: 45 %
SOR XIC B9:11/2 OTE O:11.0/2 EOR
%   B9:11/2  "ALARM 3 LOOP HIGH CONDUCTIVITY" %
%   O:11.0/2  "ALARM 3 LOOP HIGH CONDUCTIVITY" %
% Rung: 46 %
SOR XIC B9:11/3 OTE O:11.0/3 EOR
%   B9:11/3  "ALARM 4 LOOP LOW TEMPERATURE" %
%   O:11.0/3  "ALARM 4 LOOP LOW TEMPERATURE" %
% Rung: 47 %
SOR XIC B9:11/4 OTE O:11.0/4 EOR
%   B9:11/4  "ALARM 5 STORAGE VESSEL LOW TEMPERATURE" %
%   O:11.0/4  "ALARM 5 STORAGE VESSEL LOW TEMPERATURE" %
% Rung: 48 %
SOR XIC B9:11/5 OTE O:11.0/5 EOR
%   B9:11/5  "ALARM 6 VESSEL HIGH LEVEL PROB/SWITH" %
%   O:11.0/5  "ALARM 6 VESSEL HIGH LEVEL PROB/SWITH" %

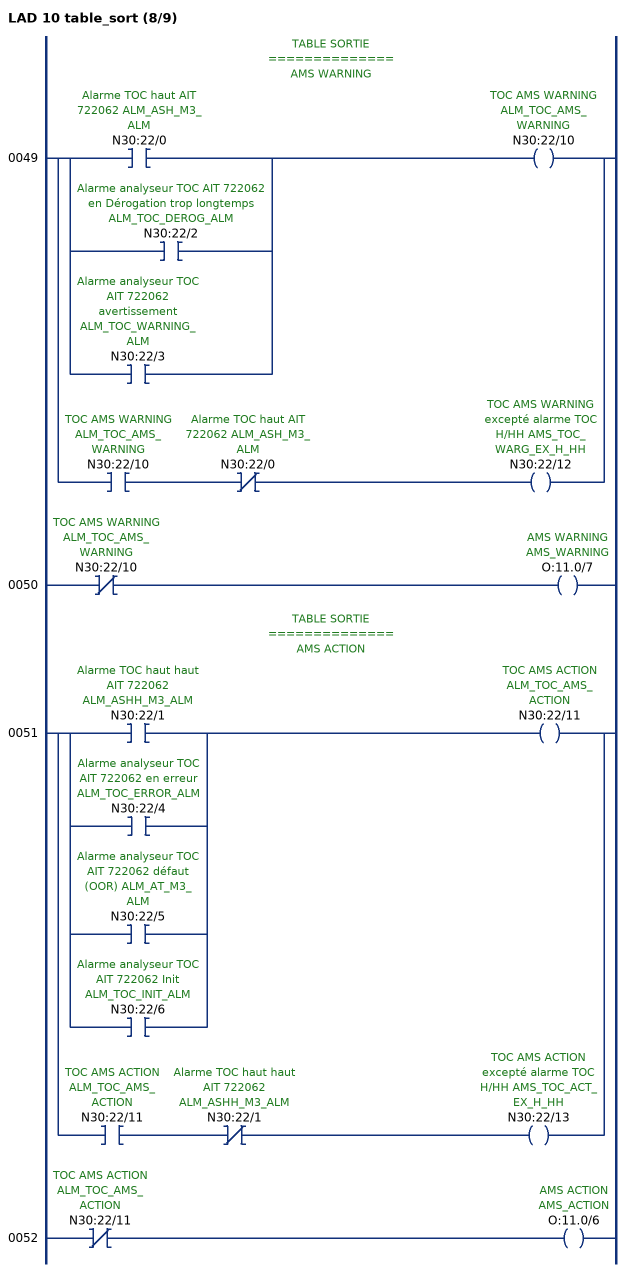
% Rung: 49 %
% TABLE SORTIE
% ==============
% AMS WARNING %
SOR BST BST XIC N30:22/0 NXB XIC N30:22/2 NXB XIC N30:22/3 BND OTE N30:22/10 NXB XIC N30:22/10 XIO N30:22/0 OTE N30:22/12 BND EOR
%   N30:22/0  ALM_ASH_M3_ALM  "Alarme TOC haut AIT 722062" %
%   N30:22/2  ALM_TOC_DEROG_ALM  "Alarme analyseur TOC AIT 722062 en Dérogation trop longtemps" %
%   N30:22/3  ALM_TOC_WARNING_ALM  "Alarme analyseur TOC AIT 722062 avertissement" %
%   N30:22/10  ALM_TOC_AMS_WARNING  "TOC AMS WARNING" %
%   N30:22/12  AMS_TOC_WARG_EX_H_HH  "TOC AMS WARNING excepté alarme TOC H/HH" %
% Rung: 50 %
SOR XIO N30:22/10 OTE O:11.0/7 EOR
%   N30:22/10  ALM_TOC_AMS_WARNING  "TOC AMS WARNING" %
%   O:11.0/7  AMS_WARNING  "AMS WARNING" %
% Rung: 51 %
% TABLE SORTIE
% ==============
% AMS ACTION %
SOR BST BST XIC N30:22/1 NXB XIC N30:22/4 NXB XIC N30:22/5 NXB XIC N30:22/6 BND OTE N30:22/11 NXB XIC N30:22/11 XIO N30:22/1 OTE N30:22/13 BND EOR
%   N30:22/1  ALM_ASHH_M3_ALM  "Alarme TOC haut haut AIT 722062" %
%   N30:22/4  ALM_TOC_ERROR_ALM  "Alarme analyseur TOC AIT 722062 en erreur" %
%   N30:22/5  ALM_AT_M3_ALM  "Alarme analyseur TOC AIT 722062 défaut (OOR)" %
%   N30:22/6  ALM_TOC_INIT_ALM  "Alarme analyseur TOC AIT 722062 Init" %
%   N30:22/11  ALM_TOC_AMS_ACTION  "TOC AMS ACTION" %
%   N30:22/13  AMS_TOC_ACT_EX_H_HH  "TOC AMS ACTION excepté alarme TOC H/HH" %
% Rung: 52 %
SOR XIO N30:22/11 OTE O:11.0/6 EOR
%   N30:22/11  ALM_TOC_AMS_ACTION  "TOC AMS ACTION" %
%   O:11.0/6  AMS_ACTION  "AMS ACTION" %

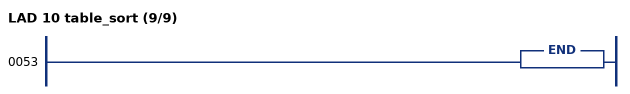
% Rung: 53 %
SOR END EOR

LADDER 29 "IN_TOC"    % TABLE ENTREE/ SOUS-ROUTINE TOC %
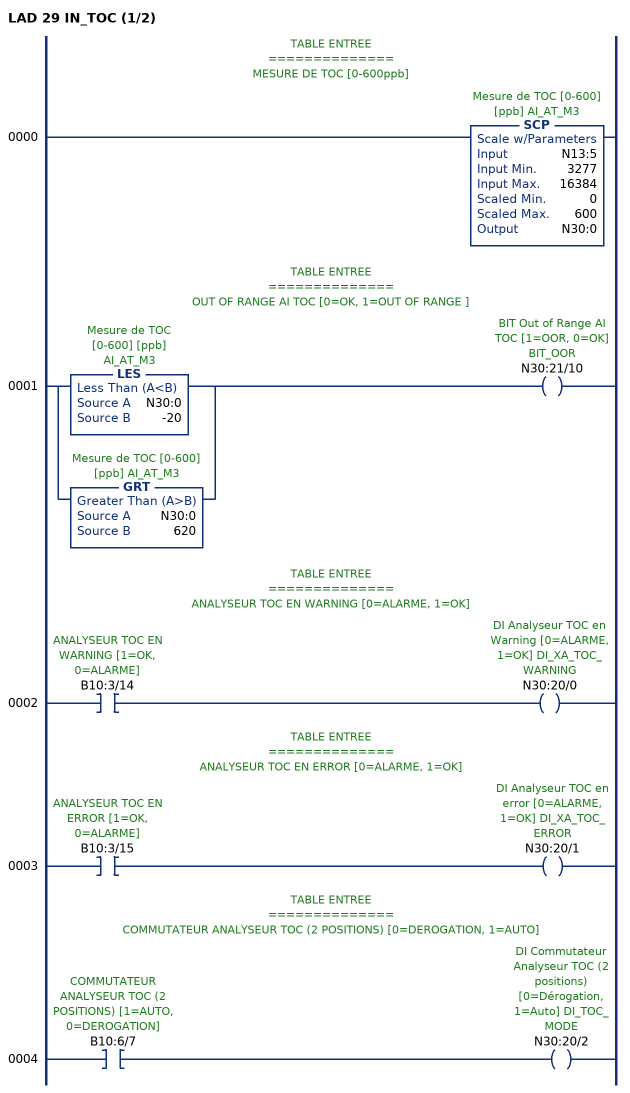
% Rung: 0 %
% TABLE ENTREE
% ==============
% MESURE DE TOC [0-600ppb] %
SOR SCP N13:5 3277 16384 0 600 N30:0 EOR
%   N13:5  AT_M3  "ANALOG IN EPI-LOOP CONDUCTIV. AIT722062" %
%   N30:0  AI_AT_M3  "Mesure de TOC [0-600] [ppb]" %
% Rung: 1 %
% TABLE ENTREE
% ==============
% OUT OF RANGE AI TOC [0=OK, 1=OUT OF RANGE ] %
SOR BST LES N30:0 -20 NXB GRT N30:0 620 BND OTE N30:21/10 EOR
%   N30:0  AI_AT_M3  "Mesure de TOC [0-600] [ppb]" %
%   N30:21/10  BIT_OOR  "BIT Out of Range AI TOC [1=OOR, 0=OK]" %
% Rung: 2 %
% TABLE ENTREE
% ==============
% ANALYSEUR TOC EN WARNING [0=ALARME, 1=OK] %
SOR XIC B10:3/14 OTE N30:20/0 EOR
%   B10:3/14  "ANALYSEUR TOC EN WARNING [1=OK, 0=ALARME]" %
%   N30:20/0  DI_XA_TOC_WARNING  "DI Analyseur TOC en Warning [0=ALARME, 1=OK]" %
% Rung: 3 %
% TABLE ENTREE
% ==============
% ANALYSEUR TOC EN ERROR [0=ALARME, 1=OK] %
SOR XIC B10:3/15 OTE N30:20/1 EOR
%   B10:3/15  "ANALYSEUR TOC EN ERROR [1=OK, 0=ALARME]" %
%   N30:20/1  DI_XA_TOC_ERROR  "DI Analyseur TOC en error [0=ALARME, 1=OK]" %
% Rung: 4 %
% TABLE ENTREE
% ==============
% COMMUTATEUR ANALYSEUR TOC (2 POSITIONS) [0=DEROGATION, 1=AUTO] %
SOR XIC B10:6/7 OTE N30:20/2 EOR
%   B10:6/7  "COMMUTATEUR ANALYSEUR TOC (2 POSITIONS) [1=AUTO, 0=DEROGATION]" %
%   N30:20/2  DI_TOC_MODE  "DI Commutateur Analyseur TOC (2 positions) [0=Dérogation, 1=Auto]" %

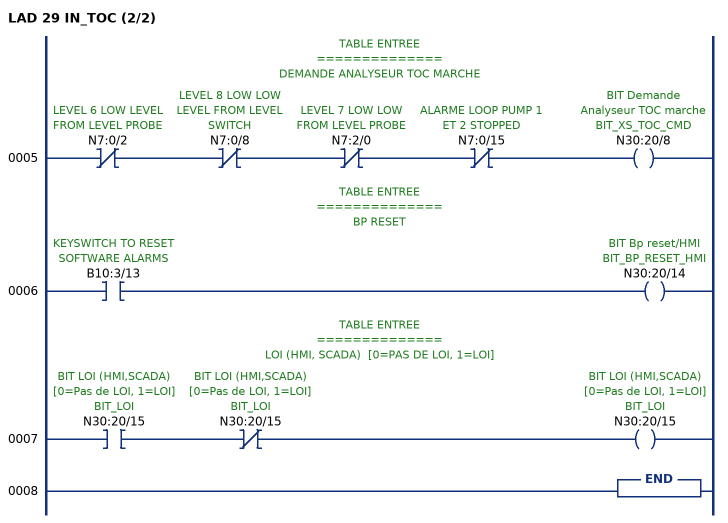
% Rung: 5 %
% TABLE ENTREE
% ==============
% DEMANDE ANALYSEUR TOC MARCHE %
SOR XIO N7:0/2 XIO N7:0/8 XIO N7:2/0 XIO N7:0/15 OTE N30:20/8 EOR
%   N7:0/2  "LEVEL 6 LOW LEVEL FROM LEVEL PROBE" %
%   N7:0/8  "LEVEL 8 LOW LOW LEVEL FROM LEVEL SWITCH" %
%   N7:2/0  "LEVEL 7 LOW LOW FROM LEVEL PROBE" %
%   N7:0/15  "ALARME LOOP PUMP 1 ET 2 STOPPED" %
%   N30:20/8  BIT_XS_TOC_CMD  "BIT Demande Analyseur TOC marche" %
% Rung: 6 %
% TABLE ENTREE
% ==============
% BP RESET %
SOR XIC B10:3/13 OTE N30:20/14 EOR
%   B10:3/13  "KEYSWITCH TO RESET SOFTWARE ALARMS" %
%   N30:20/14  BIT_BP_RESET_HMI  "BIT Bp reset/HMI" %
% Rung: 7 %
% TABLE ENTREE
% ==============
% LOI (HMI, SCADA)  [0=PAS DE LOI, 1=LOI] %
SOR XIC N30:20/15 XIO N30:20/15 OTE N30:20/15 EOR
%   N30:20/15  BIT_LOI  "BIT LOI (HMI,SCADA) [0=Pas de LOI, 1=LOI]" %
% Rung: 8 %
SOR END EOR

LADDER 30 "TOC"    % SOUS-ROUTINE TOC %
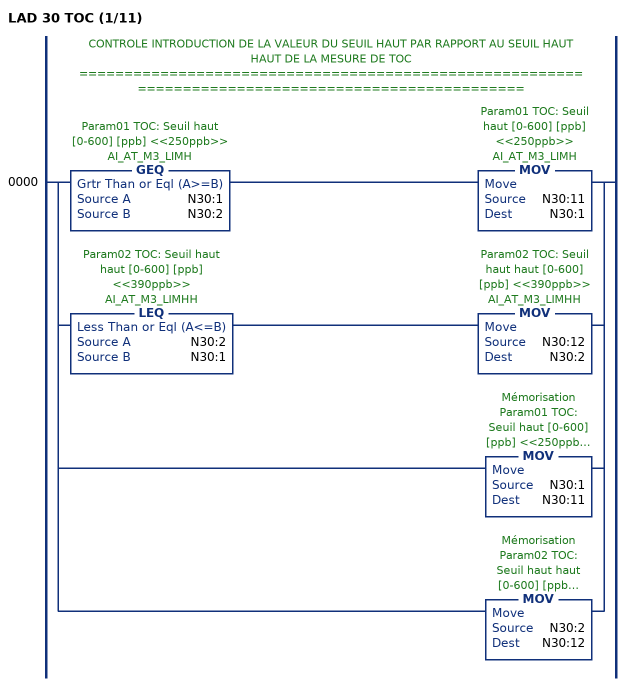
% Rung: 0 %
% CONTROLE INTRODUCTION DE LA VALEUR DU SEUIL HAUT PAR RAPPORT AU SEUIL HAUT HAUT DE LA MESURE DE TOC
% =================================================================================================== %
SOR BST GEQ N30:1 N30:2 MOV N30:11 N30:1 NXB LEQ N30:2 N30:1 MOV N30:12 N30:2 NXB MOV N30:1 N30:11 NXB MOV N30:2 N30:12 BND EOR
%   N30:1  AI_AT_M3_LIMH  "Param01 TOC: Seuil haut [0-600] [ppb] <<250ppb>>" %
%   N30:2  AI_AT_M3_LIMHH  "Param02 TOC: Seuil haut haut [0-600] [ppb] <<390ppb>>" %
%   N30:11  MEMO_AT_M3_LIMH  "Mémorisation Param01 TOC: Seuil haut [0-600] [ppb] <<250ppb>>" %
%   N30:12  MEMO_AT_M3_LIMHH  "Mémorisation Param02 TOC: Seuil haut haut [0-600] [ppb] <<500ppb>>" %

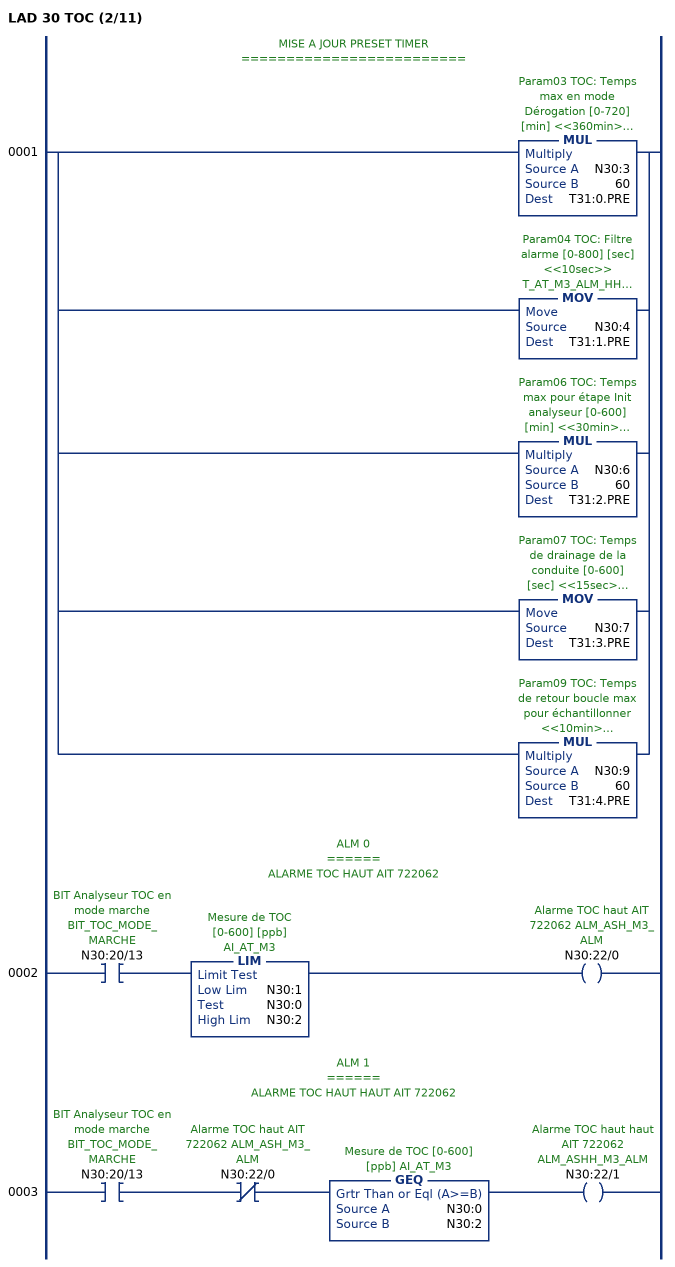
% Rung: 1 %
% MISE A JOUR PRESET TIMER
% ========================= %
SOR BST MUL N30:3 60 T31:0.PRE NXB MOV N30:4 T31:1.PRE NXB MUL N30:6 60 T31:2.PRE NXB MOV N30:7 T31:3.PRE NXB MUL N30:9 60 T31:4.PRE BND EOR
%   N30:3  AI_TOC_DEROG_LIMH  "Param03 TOC: Temps max en mode Dérogation [0-960] [min] <<360min>>" %
%   T31:0  T_TOC_DEROG_LIMH  "Param03 TOC: Temps max en mode Dérogation [0-720] [min] <<360min>>" %
%   N30:4  AI_AT_M3_ALM_HH_DL  "Param04 TOC: Filtre alarme [0-800] [sec] <<10sec>>" %
%   T31:1  T_AT_M3_ALM_HH_DL  "Param04 TOC: Filtre alarme [0-800] [sec] <<10sec>>" %
%   N30:6  AI_TOC_INIT_LIMH  "Param06 TOC: Temps max pour étape Init analyseur [0-600] [min] <<30min>>" %
%   T31:2  T_TOC_INIT_LIMH  "Param06 TOC: Temps max pour étape Init analyseur [0-600] [min] <<30min>>" %
%   N30:7  AI_XV_M3_CMD_DELAY  "Param07 TOC: Temps de drainage de la conduite [0-600] [sec] <<15sec>>" %
%   T31:3  T_XV_M3_CMD_DELAY  "Param07 TOC: Temps de drainage de la conduite [0-600] [sec] <<15sec>>" %
%   N30:9  AI_T_TT_722011_LIMH  "Param09 TOC: Temps filtrage sur Température retour boucle [] [min] <<10 min>>" %
%   T31:4  T_TT_722011_LIMH  "Param09 TOC: Temps de retour boucle max pour échantillonner <<10min>>" %
% Rung: 2 %
% ALM 0
% ======
% ALARME TOC HAUT AIT 722062 %
SOR XIC N30:20/13 LIM N30:1 N30:0 N30:2 OTE N30:22/0 EOR
%   N30:20/13  BIT_TOC_MODE_MARCHE  "BIT Analyseur TOC en mode marche" %
%   N30:1  AI_AT_M3_LIMH  "Param01 TOC: Seuil haut [0-600] [ppb] <<250ppb>>" %
%   N30:0  AI_AT_M3  "Mesure de TOC [0-600] [ppb]" %
%   N30:2  AI_AT_M3_LIMHH  "Param02 TOC: Seuil haut haut [0-600] [ppb] <<390ppb>>" %
%   N30:22/0  ALM_ASH_M3_ALM  "Alarme TOC haut AIT 722062" %
% Rung: 3 %
% ALM 1
% ======
% ALARME TOC HAUT HAUT AIT 722062 %
SOR XIC N30:20/13 XIO N30:22/0 GEQ N30:0 N30:2 OTE N30:22/1 EOR
%   N30:20/13  BIT_TOC_MODE_MARCHE  "BIT Analyseur TOC en mode marche" %
%   N30:22/0  ALM_ASH_M3_ALM  "Alarme TOC haut AIT 722062" %
%   N30:0  AI_AT_M3  "Mesure de TOC [0-600] [ppb]" %
%   N30:2  AI_AT_M3_LIMHH  "Param02 TOC: Seuil haut haut [0-600] [ppb] <<390ppb>>" %
%   N30:22/1  ALM_ASHH_M3_ALM  "Alarme TOC haut haut AIT 722062" %

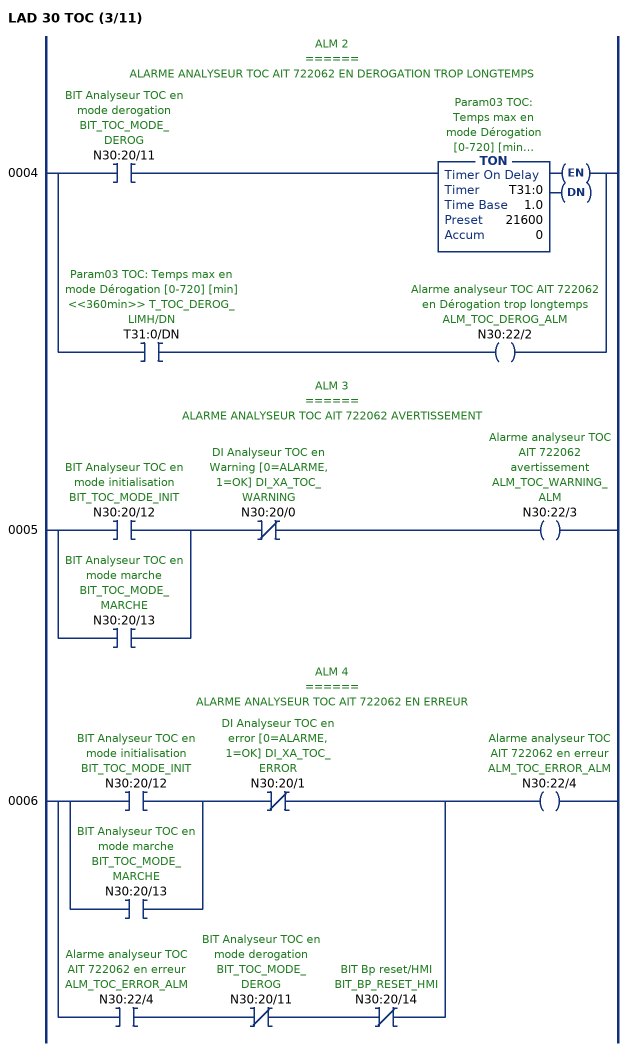
% Rung: 4 %
% ALM 2
% ======
% ALARME ANALYSEUR TOC AIT 722062 EN DEROGATION TROP LONGTEMPS %
SOR BST XIC N30:20/11 TON T31:0 1.0 21600 0 NXB XIC T31:0/DN OTE N30:22/2 BND EOR
%   N30:20/11  BIT_TOC_MODE_DEROG  "BIT Analyseur TOC en mode derogation" %
%   T31:0  T_TOC_DEROG_LIMH  "Param03 TOC: Temps max en mode Dérogation [0-720] [min] <<360min>>" %
%   N30:22/2  ALM_TOC_DEROG_ALM  "Alarme analyseur TOC AIT 722062 en Dérogation trop longtemps" %
% Rung: 5 %
% ALM 3
% ======
% ALARME ANALYSEUR TOC AIT 722062 AVERTISSEMENT %
SOR BST XIC N30:20/12 NXB XIC N30:20/13 BND XIO N30:20/0 OTE N30:22/3 EOR
%   N30:20/12  BIT_TOC_MODE_INIT  "BIT Analyseur TOC en mode initialisation" %
%   N30:20/13  BIT_TOC_MODE_MARCHE  "BIT Analyseur TOC en mode marche" %
%   N30:20/0  DI_XA_TOC_WARNING  "DI Analyseur TOC en Warning [0=ALARME, 1=OK]" %
%   N30:22/3  ALM_TOC_WARNING_ALM  "Alarme analyseur TOC AIT 722062 avertissement" %
% Rung: 6 %
% ALM 4
% ======
% ALARME ANALYSEUR TOC AIT 722062 EN ERREUR %
SOR BST BST XIC N30:20/12 NXB XIC N30:20/13 BND XIO N30:20/1 NXB XIC N30:22/4 XIO N30:20/11 XIO N30:20/14 BND OTE N30:22/4 EOR
%   N30:20/12  BIT_TOC_MODE_INIT  "BIT Analyseur TOC en mode initialisation" %
%   N30:20/13  BIT_TOC_MODE_MARCHE  "BIT Analyseur TOC en mode marche" %
%   N30:20/1  DI_XA_TOC_ERROR  "DI Analyseur TOC en error [0=ALARME, 1=OK]" %
%   N30:22/4  ALM_TOC_ERROR_ALM  "Alarme analyseur TOC AIT 722062 en erreur" %
%   N30:20/11  BIT_TOC_MODE_DEROG  "BIT Analyseur TOC en mode derogation" %
%   N30:20/14  BIT_BP_RESET_HMI  "BIT Bp reset/HMI" %

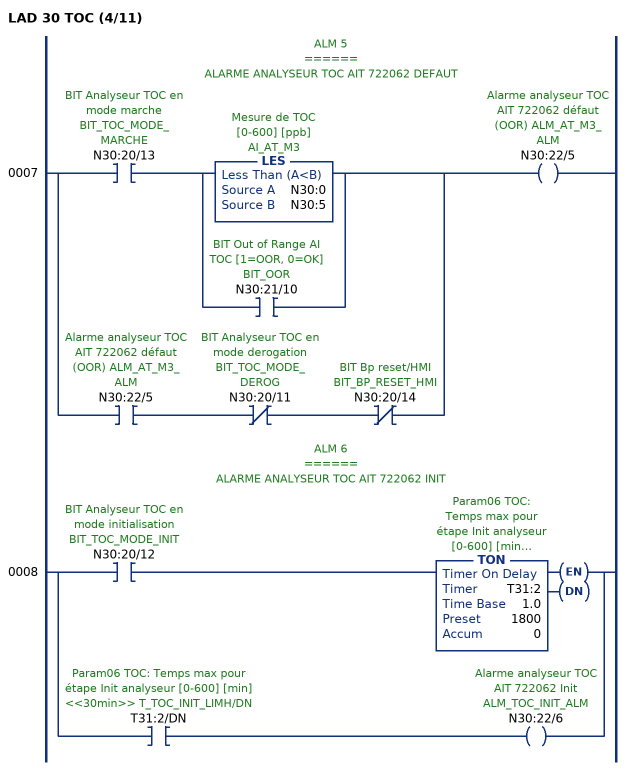
% Rung: 7 %
% ALM 5
% ======
% ALARME ANALYSEUR TOC AIT 722062 DEFAUT %
SOR BST XIC N30:20/13 BST LES N30:0 N30:5 NXB XIC N30:21/10 BND NXB XIC N30:22/5 XIO N30:20/11 XIO N30:20/14 BND OTE N30:22/5 EOR
%   N30:20/13  BIT_TOC_MODE_MARCHE  "BIT Analyseur TOC en mode marche" %
%   N30:0  AI_AT_M3  "Mesure de TOC [0-600] [ppb]" %
%   N30:5  AI_AT_M3_MIN  "Param05 TOC: Seuil d'initialisation de mesure de TOC [0-600] [ppb] <<4ppb>>" %
%   N30:21/10  BIT_OOR  "BIT Out of Range AI TOC [1=OOR, 0=OK]" %
%   N30:22/5  ALM_AT_M3_ALM  "Alarme analyseur TOC AIT 722062 défaut (OOR)" %
%   N30:20/11  BIT_TOC_MODE_DEROG  "BIT Analyseur TOC en mode derogation" %
%   N30:20/14  BIT_BP_RESET_HMI  "BIT Bp reset/HMI" %
% Rung: 8 %
% ALM 6
% ======
% ALARME ANALYSEUR TOC AIT 722062 INIT %
SOR BST XIC N30:20/12 TON T31:2 1.0 1800 0 NXB XIC T31:2/DN OTE N30:22/6 BND EOR
%   N30:20/12  BIT_TOC_MODE_INIT  "BIT Analyseur TOC en mode initialisation" %
%   T31:2  T_TOC_INIT_LIMH  "Param06 TOC: Temps max pour étape Init analyseur [0-600] [min] <<30min>>" %
%   N30:22/6  ALM_TOC_INIT_ALM  "Alarme analyseur TOC AIT 722062 Init" %

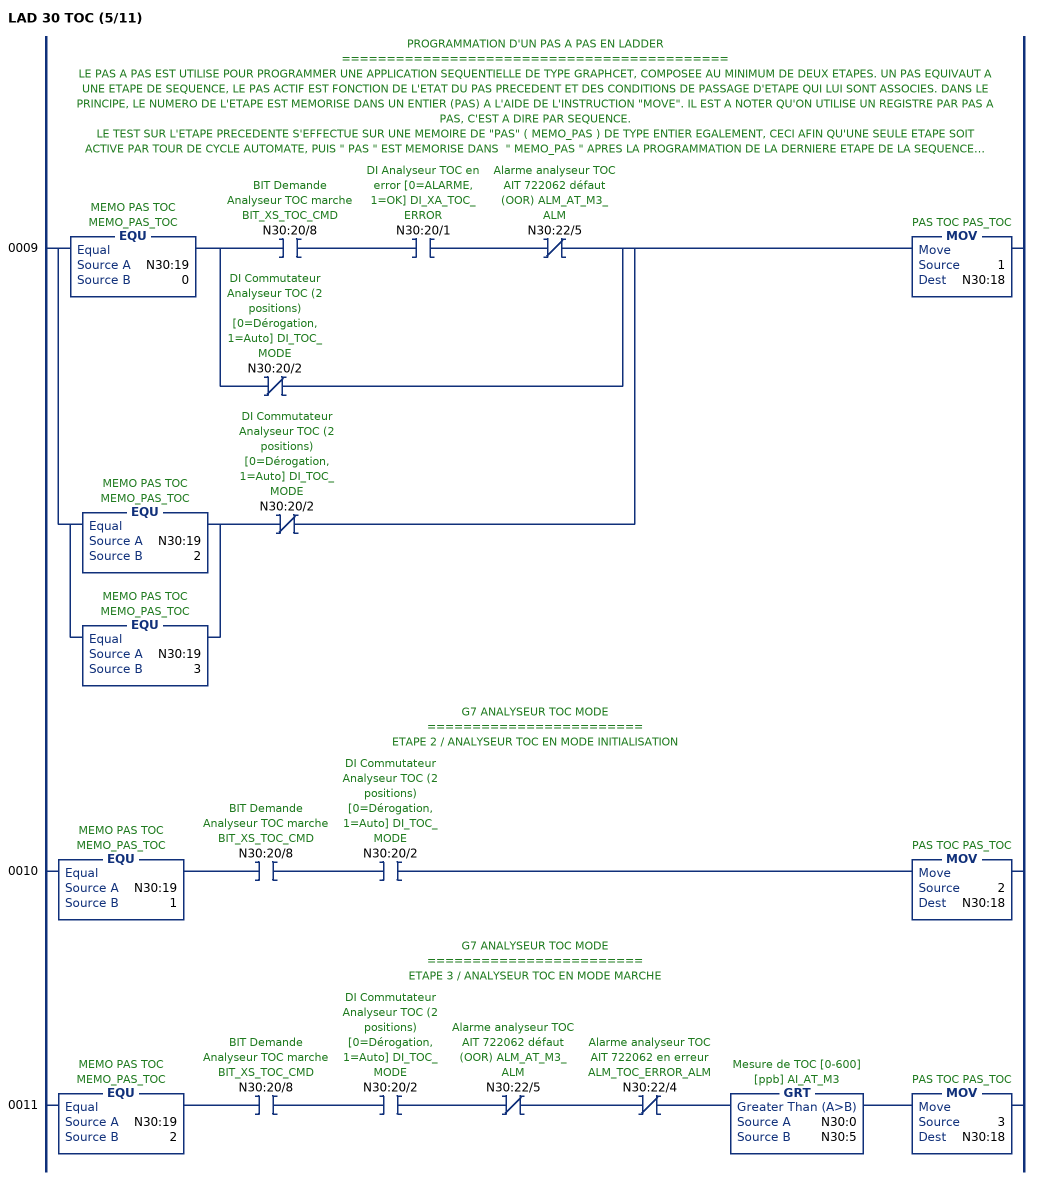
% Rung: 9 %
% PROGRAMMATION D'UN PAS A PAS EN LADDER
% ===========================================
% LE PAS A PAS EST UTILISE POUR PROGRAMMER UNE APPLICATION SEQUENTIELLE DE TYPE GRAPHCET, COMPOSEE AU MINIMUM DE DEUX ETAPES. UN PAS EQUIVAUT A UNE ETAPE DE SEQUENCE, LE PAS ACTIF EST FONCTION DE L'ETAT DU PAS PRECEDENT ET DES CONDITIONS DE PASSAGE D'ETAPE QUI LUI SONT ASSOCIES. DANS LE PRINCIPE, LE NUMERO DE L'ETAPE EST MEMORISE DANS UN ENTIER (PAS) A L'AIDE DE L'INSTRUCTION "MOVE". IL EST A NOTER QU'ON UTILISE UN REGISTRE PAR PAS A PAS, C'EST A DIRE PAR SEQUENCE.
% LE TEST SUR L'ETAPE PRECEDENTE S'EFFECTUE SUR UNE MEMOIRE DE "PAS" ( MEMO_PAS ) DE TYPE ENTIER EGALEMENT, CECI AFIN QU'UNE SEULE ETAPE SOIT ACTIVE PAR TOUR DE CYCLE AUTOMATE, PUIS " PAS " EST MEMORISE DANS  " MEMO_PAS " APRES LA PROGRAMMATION DE LA DERNIERE ETAPE DE LA SEQUENCE.
% 
% G7 ANALYSEUR TOC MODE
% ========================
% ETAPE 1 / ANALYSEUR TOC EN MODE DEROGATION %
SOR BST EQU N30:19 0 BST XIC N30:20/8 XIC N30:20/1 XIO N30:22/5 NXB XIO N30:20/2 BND NXB BST EQU N30:19 2 NXB EQU N30:19 3 BND XIO N30:20/2 BND MOV 1 N30:18 EOR
%   N30:19  MEMO_PAS_TOC  "MEMO PAS TOC" %
%   N30:20/8  BIT_XS_TOC_CMD  "BIT Demande Analyseur TOC marche" %
%   N30:20/1  DI_XA_TOC_ERROR  "DI Analyseur TOC en error [0=ALARME, 1=OK]" %
%   N30:22/5  ALM_AT_M3_ALM  "Alarme analyseur TOC AIT 722062 défaut (OOR)" %
%   N30:20/2  DI_TOC_MODE  "DI Commutateur Analyseur TOC (2 positions) [0=Dérogation, 1=Auto]" %
%   N30:18  PAS_TOC  "PAS TOC" %
% Rung: 10 %
% G7 ANALYSEUR TOC MODE
% ========================
% ETAPE 2 / ANALYSEUR TOC EN MODE INITIALISATION %
SOR EQU N30:19 1 XIC N30:20/8 XIC N30:20/2 MOV 2 N30:18 EOR
%   N30:19  MEMO_PAS_TOC  "MEMO PAS TOC" %
%   N30:20/8  BIT_XS_TOC_CMD  "BIT Demande Analyseur TOC marche" %
%   N30:20/2  DI_TOC_MODE  "DI Commutateur Analyseur TOC (2 positions) [0=Dérogation, 1=Auto]" %
%   N30:18  PAS_TOC  "PAS TOC" %
% Rung: 11 %
% G7 ANALYSEUR TOC MODE
% ========================
% ETAPE 3 / ANALYSEUR TOC EN MODE MARCHE %
SOR EQU N30:19 2 XIC N30:20/8 XIC N30:20/2 XIO N30:22/5 XIO N30:22/4 GRT N30:0 N30:5 MOV 3 N30:18 EOR
%   N30:19  MEMO_PAS_TOC  "MEMO PAS TOC" %
%   N30:20/8  BIT_XS_TOC_CMD  "BIT Demande Analyseur TOC marche" %
%   N30:20/2  DI_TOC_MODE  "DI Commutateur Analyseur TOC (2 positions) [0=Dérogation, 1=Auto]" %
%   N30:22/5  ALM_AT_M3_ALM  "Alarme analyseur TOC AIT 722062 défaut (OOR)" %
%   N30:22/4  ALM_TOC_ERROR_ALM  "Alarme analyseur TOC AIT 722062 en erreur" %
%   N30:0  AI_AT_M3  "Mesure de TOC [0-600] [ppb]" %
%   N30:5  AI_AT_M3_MIN  "Param05 TOC: Seuil d'initialisation de mesure de TOC [0-600] [ppb] <<4ppb>>" %
%   N30:18  PAS_TOC  "PAS TOC" %

